PROGRAM ChargeTime
VAR

	//lca_charge_cal	 : ARRAY [1..6] OF LCA_CAL;
	i				 : INT := 1; // 1-6 instances
	j				 : INT := 1; //1 - 6 ch
	m				 : INT := 1;
	n				 : INT := 6;
	a				 : INT := 1; 
	
	Q				 : REAL := 1; // Charge
	Current			 : REAL := 0.1; //100mA
	
	longestChargeTime: REAL;
	
END_VAR

//mapping hmi input to setpoints
FOR j := 1 TO n BY 1 DO	
	Setpoints.HPT5[j].TotalCapacitance	:= HMI_DB.HPT5[j].TotalCapacitance;
	//Setpoints.TDKLoad[j].PSratedV 			:= HMI_DB.TDKLoad[j].PSratedV;
	Setpoints.HPT5[j].RequiredChargedV	:= HMI_DB.HPT5[j].RequiredChargedV;  
	//Setpoints.TDKLoad[j].wLCA				:= HMI_DB.TDKLoad[j].wLCA;
	//Setpoints.TDKLoad[j].NumOfCharger		:= HMI_DB.TDKLoad[j].NumOfCharger;	
	
	//charge time delay and elapse for HMI
	ChargeTime_DB.ChargeTimeStartDelay[j] := TIME_TO_INT((ChargeTime_DB.ChargerDelay_PT[j] - ChargeTime_DB.ChargerDelay_ET[j])/1000);
	ChargeTime_DB.ChargingTimeElapse[j] := TIME_TO_INT((ChargeTime_DB.ChargingTimeElapse_TON[j].PT - ChargeTime_DB.ChargingTimeElapse_TON[j].ET)/1000);
END_FOR


//ChargeTime_DB.PreFormChargeTimeStartDelay := TIME_TO_INT((ChargeTime_DB.PreFormChargeTime_PT - ChargeTime_DB.PreFormChargeTime_ET)/1000);
//ChargeTime_DB.PreFormChargingTimeElapse := TIME_TO_INT((ChargeTime_DB.PreFormChargingTimeElapse_TON.PT - ChargeTime_DB.PreFormChargingTimeElapse_TON.ET)/1000);

(*
//GLS 3
Setpoints.GLSLoad.TotalCapacitance	:= HMI_DB.GLSLoad.TotalCapacitance;
Setpoints.GLSLoad.PSratedV 			:= HMI_DB.GLSLoad.PSratedV;
//Setpoints.PreFormBank.RequiredChargedV	:= Recipe.PreFormBank.RequiredChargedV; //only thing that comes from the main plc recipe
//Setpoints.GLSLoad.wLCA				:= HMI_DB.GLSLoad.wLCA;
Setpoints.GLSLoad.NumOfCharger		:= HMI_DB.GLSLoad.NumOfCharger;	
*)


//veto
//this should not happen
FOR m := 1 TO n BY 1 DO
	IF Setpoints.HPT5[m].RequiredChargedV <= -1 THEN
		Setpoints.HPT5[m].RequiredChargedV := 0;
	END_IF	
END_FOR

FOR i := 1 TO n BY 1 DO
	//set limites of charger voltage input from HMI input
	IF (Setpoints.HPT5[i].RequiredChargedV) >= AnalogConversion.MaxVolt THEN
		Setpoints.HPT5[i].RequiredChargedV := AnalogConversion.MaxVolt; //limit at 105v
		HMI_DB.HPT5[i].RequiredChargedV := AnalogConversion.MaxVolt;
	ELSIF Setpoints.HPT5[i].RequiredChargedV <= 0 THEN
		Setpoints.HPT5[i].RequiredChargedV := 0;
		HMI_DB.HPT5[i].RequiredChargedV := 0;
	END_IF	
END_FOR;

//chg time
FOR i := 1 TO n BY 1 DO
	//manually enter charge time*********************
	MCP_IO.Charger[i].ChargeTime.timeToChargeLoad := HMI_DB.HPT5[i].ChargeTime;
	
	IF Setpoints.HPT5[i].RequiredChargedV = 0 THEN
		MCP_IO.Charger[i].ChargeTime.timeToChargeLoad := 0;
		MCP_IO.Charger[i].ChargeTime.Power := 0;
	END_IF
END_FOR

(*
//gls - gls3 is preform cap charger
Q := 1000* Setpoints.GLSLoad.RequiredChargedV * (Setpoints.GLSLoad.TotalCapacitance / 1000000);
MCP_IO.GLS3_Load.timeToChargeLoad := Q / Current;
MCP_IO.GLS3_Load.Power := 1000*Setpoints.GLSLoad.RequiredChargedV * Current;
*)

//find the longest charge time.  //need more work
longestChargeTime := MAX( MCP_IO.Charger[1].ChargeTime.timeToChargeLoad,
							MCP_IO.Charger[2].ChargeTime.timeToChargeLoad,
							MCP_IO.Charger[3].ChargeTime.timeToChargeLoad,
							MCP_IO.Charger[4].ChargeTime.timeToChargeLoad,
							MCP_IO.Charger[5].ChargeTime.timeToChargeLoad,
							MCP_IO.Charger[6].ChargeTime.timeToChargeLoad);

ChargeTime_DB.LongestChargeTime_PT := REAL_TO_TIME (1000*longestChargeTime);

plc_plc_comm_DB.ChargeTime := longestChargeTime; //send charge time to m1 pp

//FOR a := 1 TO 8 BY 1 DO
FOR a := 1 TO n BY 1 DO
	IF (longestChargeTime - MCP_IO.Charger[a].ChargeTime.timeToChargeLoad) >= 0 THEN
		ChargeTime_DB.ChargerDelay_PT[a] := REAL_TO_TIME (1000*(longestChargeTime - MCP_IO.Charger[a].ChargeTime.timeToChargeLoad));
		ELSE 
			ChargeTime_DB.ChargerDelay_PT[a] := REAL_TO_TIME (1000*(MCP_IO.Charger[a].ChargeTime.timeToChargeLoad - longestChargeTime));
	END_IF;		
		
	//IF (longestChargeTime - MCP_IO.Charger[a+3].ChargeTime.timeToChargeLoad) >= 0 THEN
	//	ChargeTime_DB.SustChargeTime_PT[a] := REAL_TO_TIME (1000*(longestChargeTime - MCP_IO.Charger[a+3].ChargeTime.timeToChargeLoad));	
	//END_IF;	
	
END_FOR;


(*IF (longestChargeTime - MCP_IO.Charger[7].ChargeTime.timeToChargeLoad) >= 0 THEN
	ChargeTime_DB.FormChargeTime_PT[1] := REAL_TO_TIME (1000*(longestChargeTime - MCP_IO.Charger[7].ChargeTime.timeToChargeLoad));	
END_IF;	
IF (longestChargeTime - MCP_IO.Charger[8].ChargeTime.timeToChargeLoad) >= 0 THEN
	ChargeTime_DB.FormChargeTime_PT[2] := REAL_TO_TIME (1000*(longestChargeTime - MCP_IO.Charger[8].ChargeTime.timeToChargeLoad));	
END_IF;	

IF (longestChargeTime - MCP_IO.GLS3_Load.timeToChargeLoad) >= 0 THEN
		ChargeTime_DB.PreFormChargeTime_PT := REAL_TO_TIME (1000*(longestChargeTime - MCP_IO.GLS3_Load.timeToChargeLoad));
		ELSE
			ChargeTime_DB.PreFormChargeTime_PT := REAL_TO_TIME (1000*(MCP_IO.GLS3_Load.timeToChargeLoad -longestChargeTime));
END_IF;
*)



IF i > n THEN 
	i := 1;
END_IF

IF j > n THEN
	j := 1;
END_IF

IF m > n THEN
	m := 1;
END_IF


IF a > n THEN
	a := 1;
END_IF;

END_PROGRAM

(* stored: Version 1.1.0.1, ProductVersion 3.1.4024.11
   POU ChargeTime: Id {28824270-3930-44b7-bfe2-d4b07042cd6b}, SpecialFunc None *)
